# EPICS StreamDevice protocol: docker/stream/PS_DB/tc-l2s.proto
Terminator = CR LF;
MaxInput=5;
getDOR {
  out "@DOR?";
  in "%5c";
}
